SUBAPPLICATION mapping_aux (* Subapplication Type *)
  (* Standard: 61499-2 *)
  (* Version 1.0, 2023-01-29, Franz *)
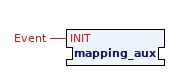
  EVENT_INPUT
    INIT;
  END_EVENT
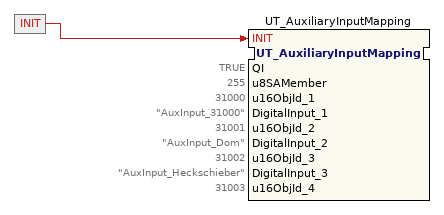
  FBS
    UT_AuxiliaryInputMapping : UT_AuxiliaryInputMapping(QI := TRUE, u8SAMember := 255, u16ObjId_1 := 31000, DigitalInput_1 := "AuxInput_31000", u16ObjId_2 := 31001, DigitalInput_2 := "AuxInput_Dom", u16ObjId_3 := 31002, DigitalInput_3 := "AuxInput_Heckschieber", u16ObjId_4 := 31003);
  END_FBS
  EVENT_CONNECTIONS
    INIT TO UT_AuxiliaryInputMapping.INIT;
  END_CONNECTIONS
END_SUBAPPLICATION
